FUNCTION_BLOCK BasicCalcManyStates (* Basic FB with empty ECC *)
  (* Standard: 61499-2 *)
  (* Version 1.0, 2023-07-26, AK115394 *)
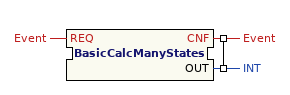
  EVENT_INPUT
    REQ;
  END_EVENT
  EVENT_OUTPUT
    CNF WITH OUT;
  END_EVENT
  VAR_OUTPUT
    OUT : INT;
  END_VAR
  VAR
    Fn0 : INT;
    Fn1 : INT;
    Fnx : INT;
  END_VAR
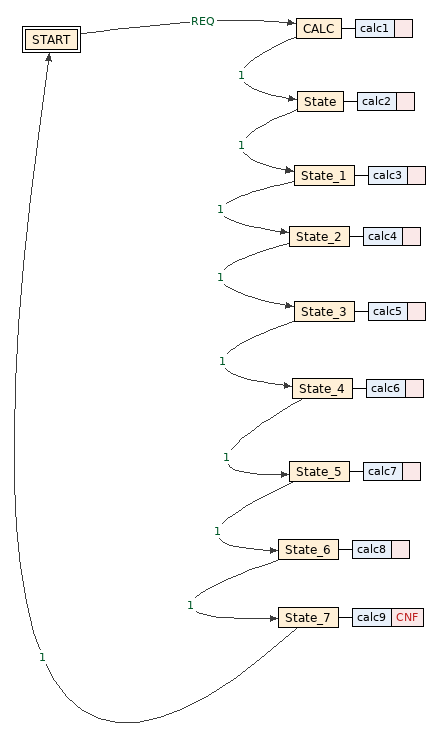
  EC_STATES
    START; (* Initial State *)
    CALC : calc1;
    State : calc2;
    State_1 : calc3;
    State_2 : calc4;
    State_3 : calc5;
    State_4 : calc6;
    State_5 : calc7;
    State_6 : calc8;
    State_7 : calc9 -> CNF;
  END_STATES
  EC_TRANSITIONS
    START TO CALC := REQ;
    CALC TO State := 1;
    State TO State_1 := 1;
    State_1 TO State_2 := 1;
    State_2 TO State_3 := 1;
    State_3 TO State_4 := 1;
    State_4 TO State_5 := 1;
    State_5 TO State_6 := 1;
    State_6 TO State_7 := 1;
    State_7 TO START := 1;
  END_TRANSITIONS
  ALGORITHM calc1 IN ST:
 OUT:=1+1;
  END_ALGORITHM
  ALGORITHM calc2 IN ST:
 OUT:=2+2;
  END_ALGORITHM
  ALGORITHM calc3 IN ST:
 OUT:=3+3;
  END_ALGORITHM
  ALGORITHM calc4 IN ST:
 OUT:=4+4;
  END_ALGORITHM
  ALGORITHM calc5 IN ST:
 OUT:=5+5;
  END_ALGORITHM
  ALGORITHM calc6 IN ST:
 OUT:=6+6;
  END_ALGORITHM
  ALGORITHM calc7 IN ST:
 OUT:=7+7;
  END_ALGORITHM
  ALGORITHM calc8 IN ST:
 OUT:=8+8;
  END_ALGORITHM
  ALGORITHM calc9 IN ST:
 OUT:=9+9;
  END_ALGORITHM
END_FUNCTION_BLOCK
